Universal Robots PolyScope program: buffer_test_segunda.urp

Program buffer_test_segunda (installation=botross directory=/programs/APS2OsUltimosRomanticos createdIn=3.15.3.106223 lastSavedIn=3.15.3.106223 robotSerialNumber=2017357017)
Calibrated DH parameters: a=[0.0001, -0.032836, -0.39033, 0.000086, 0.000053, 0]; d=[0.089393, 264.548863, -261.578988, -2.85966, 0.094927, 0.082356]; alpha=[1.569373, -0.001603, 0.013671, 1.570599, -1.570158, 0]; deltaTheta=[0.000031, -1.49356, 1.597104, -0.103695, -0.000023, -0.000043]
BeforeStart
  SocketIP := socket_open("10.103.16.140",30000,"gio")
  MoveJ speed 60 deg/s, acceleration 80 deg/s^2 (useActiveTCP=true)
    Waypoint origem: TCP in base x=536.622 y=-323.282 z=-120.683 mm, rx=-0.081 ry=0.0108 rz=0.1119 rad; joints [140.297, -53.428, 101.844, -140.967, -93.47, 44.531] deg; flange x=538.034 y=-308.609 z=58.713 mm, rx=0.1749 ry=-3.1217 rz=0.1268 rad
Robot Program (runOnlyOnce=false)
  Loop While (checkContinuously=false) expression=SocketIP≟ False
    SocketIP := socket_open("10.103.16.140",30000,"gio")
    Wait Sleep waitTime=0.5
    Call Rotina_Contornos
SubProgram -> Rotina_Contornos
SubProgram Rotina_Pick_Caneta (keepSynchronizedWithDisk=false)
  Wait Sleep waitTime=0.01
  'a linha a seguir causa um movimento brusco e intenso'
  Script: speedl([0.5,0.5,0.5,0,0,0],0.5,5)
SubProgram Rotina_Contornos (keepSynchronizedWithDisk=false)
  Script: socket_send_string("asking_for_data")
  Wait Sleep waitTime=0.5
  read_ascii := socket_read_ascii_float(3,"gio")
  var_1 := socket_read_ascii_float(3,"gio")
  Wait Sleep waitTime=0.5
  SocketIP := False
  Script: socket_close("gio")
  If read_ascii[0]≠0
    pose_desejada := p[read_ascii[1]/1000,read_ascii[2]/1000,var_1[1]/1000,0,0,0]
    pose_atual := get_actual_tcp_pose()
    destino := pose_trans(Plano_BotRoss,pose_desejada)
    MoveL speed 250 mm/s, acceleration 1200 mm/s^2 (useActiveTCP=true) feature=Base
      Waypoint Waypoint (Variable): variable=destino
      Wait NoWait
